FUNCTION_BLOCK FB_RV_les
VAR_INPUT
	Stellung	: REAL;
END_VAR
VAR_OUTPUT
END_VAR
VAR
	{attribute 'OPC.UA.DA' := '1'}Stellwert	: ST_RV_les_Stellwert;	
	{attribute 'OPC.UA.DA' := '1'}Zustand		: ST_RV_les_Zustand;
END_VAR
VAR // added by the converter: edge detectors and wires of the graphical bodies
    _w1 : ANY;
END_VAR

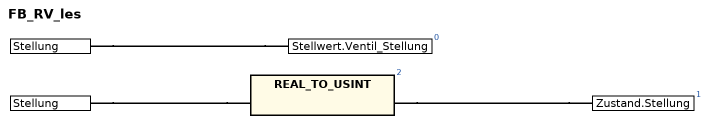
Stellwert.Ventil_Stellung := Stellung;
Zustand.Stellung := _w1;
_w1 := REAL_TO_USINT(Stellung);

END_FUNCTION_BLOCK

(* stored: Version 1.1.0.1, ProductVersion 3.1.4024.9
   POU FB_RV_les: Id {1eb84745-1db9-4332-8294-569a8c70313e}, SpecialFunc None *)
